{attribute 'GeneratedUsingTerminal: EL9930-0000-0016'}
{attribute addProperty BoxType "EL9930-0000-0016"}
{attribute addProperty Id "A_0002_EL9930_0001_0016EL9930_2CDB4CAF4A_0003_EL9930_0000_0017A_0003_EL9930_0000_0017_624233994"}
{attribute addProperty CRC "1245532711"}
{attribute addProperty Size "8"}
TYPE A_0001_EL9930_0000_0016_4A3D5227 EXTENDS EL9930_E3B075C4 :
STRUCT
	{attribute addProperty Name "A_0002_EL9930_0001_0016"}
	{attribute addProperty PreviousPort "A_0001(EL9930-0000-0016) : B"}
	A_0002_EL9930_0001_0016 : EL9930_2CDB4CAF;
	{attribute addProperty Name "A_0003_EL9930_0000_0017"}
	{attribute addProperty PreviousPort "A_0002(EL9930-0001-0016) : B"}
	A_0003_EL9930_0000_0017 : A_0003_EL9930_0000_0017_62423399;
END_STRUCT
END_TYPE

(* stored: Version 1.2.0.0, ProductVersion 3.1.4024.9
   DUT A_0001_EL9930_0000_0016_4A3D5227: Id {abc5e340-0dbb-4e06-9b00-b5a9b3aca9f5} *)
